TYPE E_Test :
(
	Empty := 0,
	STOP,
	LOAD,
	PICK,
	PRINT
);
END_TYPE

(* stored: Version 1.1.0.1, ProductVersion 3.1.0.26
   DUT E_Test: Id {54fb43fa-ef24-460d-864d-245870c953ce} *)
